// TIA Portal V20 export
TYPE "UDT_FuellstandSteuern"
   STRUCT
      EINSCHALTWERT : Real;
      AUSSCHALTWERT : Real;
      VERZOEG_NIV : Real;
      SIM : Real;
      OFFSET : Real;
      GLAETTUNG : Real;
      FRG_SIM : Bool;
      Bit9 : Bool;
      Bit10 : Bool;
      Bit11 : Bool;
      Bit12 : Bool;
      Bit13 : Bool;
      Bit14 : Bool;
      Bit15 : Bool;
      Bit0 : Bool;
      Bit1 : Bool;
      Bit2 : Bool;
      Bit3 : Bool;
      Bit4 : Bool;
      Bit5 : Bool;
      Bit6 : Bool;
      Bit7 : Bool;
   END_STRUCT;
END_TYPE
